(* IEC 61131-3 sources: Dev/Dev_V200/200 (part 8) *)

(* ---- _Nh_MNU.st ---- *)
{ $ IFDEF __NH_WEB }

(*   vyhodnotenie vybrateho menu prebieha

   -  _Nh_Web_CMD (_NhCmd)         - vyvola akciu :
   -  _NhCmdAction   - co sa ma urobit po vybrati volby menu + podporne akcie (ulozi udaje z klasickej web-maker PAGE...)
   -  _NhCmdScreen   - nadefinuje objekty obrazovky + filtre a typ obrazovky (obj)

*)

//********* MNU *******************************************

VAR_GLOBAL
  aWht   : NH_TCH_WHT;
END_VAR

FUNCTION _NhFavNaz {HIDDEN}  : BOOL    // najde aktualne vybraty FAV a zapise veho nazov
   VAR_INPUT
      sav   : BOOL;
   END_VAR
   _NhFavNaz := true;
   FOR nd := 1 TO aCfg[20].rec DO
      _NhxDev(c := 20, n := nd, x:=16);
      xFav := xDev;
      IF xFav^.cx = xA^.fav THEN
         IF sav THEN
            xFav^.cf.Name := xL^.naz;
         ELSE
            xL^.naz := xFav^.cf.Name;
         END_IF;
         nd := 0;
         RETURN;
      END_IF;
   END_FOR;
   _Nh_Lang(id := 18 ,txt := ADR( xL^.naz ), zn:=20);             // oblubene
   nd := 0;
END_FUNCTION

FUNCTION _NhDefSet {HIDDEN}  : BOOL    // vzdy na zaciatku LEN na tomto mieste sa nadefinuju parametre vsetkych browsov, frame....
   VAR_INPUT
      chg      : BOOL;
   END_VAR
   _NhDefSet      := true;
   xU^.o[1]       :=  eMnH.o[1];                                   // aktivuje logo
   IF chg THEN

      xM^.set           := false;

      xUsr^.cx.LastSet  := false;
      CASE xU^.o[2].fn OF
         23:   xU^.o[2].fn := 25;   xM^.set           := true;
                                    xUsr^.cx.LastSet  := true;
         25:   xU^.o[2].fn := 23;
        ELSE   xU^.o[2].fn := 0;
      END_CASE;
   ELSIF xUsr^.cx.Set THEN
      xU^.o[2]       :=  eMnH.o[2];                               // default setup (sivy)
      IF xUsr^.cx.LastSet THEN      //OR aSys.NewDbx THEN
         xM^.set     := true;
         xU^.o[2].fn := 25;
      ELSE
         xM^.set := false;
         xU^.o[2].fn := 23;
      END_IF;
   ELSE
      xU^.o[2].cm := 0;                                              // nezobrazi sa
      xU^.o[2].fn := 0;
      xM^.set     := 0;
   END_IF;
END_FUNCTION

/// *******************************

FUNCTION _Nh_Web_CMD_Screen    : BOOL       // NADEFINUJE OBJEKTY OBRAZOVKY podla akcie od CMD
   (*
    screen sa rozlisuje podla xL^.obj
    - vytvori cistu LVL
    - nadefinuje vrchne a spodne menu
    - v naplni nazov screenu
    - naplni filter DEV (pre brows)
    - naplni filter ROM
    - prelozi nazov do vybrateho jazyka
   *)
   VAR_INPUT
      eMnu     : BOOL;
      obr      : INT;
      obj      : USINT;
      mnu      : USINT := 0;                                               // povolenie menu zmeny DSH (cislo vrchneho menu) 1,2
		n			: USINT;
   END_VAR
   _Nh_Web_CMD_Screen   := 0;
   xM^.wht        := 20;                                                   // pokusi sa najst 1 vetu podla usra
   xL^.brw        := true;
   xL^.obj        := obj;
   xL^.vis        := true;

//   _NhxUsr(u:= xA^.usr);                                                   // namapuje usra
   IF xL^.obj > 30 THEN
      xL^.dsh        := 1;
      mnu            := 0;
   ELSE
      xL^.dsh        := xUsr^.cx.brw[ xL^.obj ];
   END_IF;
   nd             := 0;                                                    // ID textu do xL^.naz

	IF xF^.cf.c > 0 AND xF^.cf.c <> 2 THEN
	   _NhxPt(c := xF^.cf.c, n := xF^.cf.n,x:=47);               				// namapuje hlavicku, napr. koli zisteniu ROM
	END_IF;

   CASE obj OF
     0:  // home page
         mnu            := 0;
         _NhDefSet();
         xL^.vaz        := 1;
         xL^.fvz        := true;
         xU^.o[3].fn   := 0;                                              // zrusi HOME
         xU^.o[8].fn   := 0;                                              // zrusi ON/OFF
         xF^.cf.c      := 3;                                               // default DEV je zon pre cely dom
         xF^.cf.n      := 1;
         xU^.n         := 0;                                               // ziadne vybrate menu
         _NhName(xName := ADR(xL^.Naz) , cf := xF^.cf.c, nd := xF^.cf.n);  //'Môj domov';
         xM^.naz        := xL^.Naz;
         xF^.dev.n[0]   := true;
         xM^.wht        := 25;                                              // pokusi sa najst 1 vetu podla usra
         xL^.dsh        := 0;
         mnu            := 0;

     1: // brow-Zoznam FAV
            nd             := 19;                                          // cislo textu v _NhLang
            xF^.dev.n[20]  := 1;
            xU^.o[2].fn    := 32;                                          // +
            xU^.o[2].cm    := 101;                                          // pridat oblubeny do zoznamu usra
            xF^.cf.c       := 20;                                               // default DEV je zon pre cely dom
            xL^.dsh        := 1;
            mnu            := 0;

     2: // brow-FVL
            _NhFavNaz();
            xF^.dev.n[0]   := 1;
            xL^.vaz        := 1;                                           // cislo vazby
//            xL^.fvz        := true;
            xF^.cf         := xA^.fav;

     3:  // brow-Quick (FAV)
            _NhFavNaz();
            xF^.dev.n[0]   := 1;
            xL^.vaz        := 1;
//            xL^.fvz        := true;
            xF^.cf         := xA^.fav;

     4: // brow-DASH (FAV)
            _NhFavNaz();
            xF^.dev.n[0]   := 1;
            xL^.vaz        := 1;
//            xL^.fvz        := true;
            xF^.cf         := xA^.fav;

     5: // brow-Rooms
            nd             := 7;
            xF^.cf.c       := 1;
            xF^.dev.n[1]   := 1;
            IF xA^.admin THEN
               xU^.o[2].fn    := 32;                                       // pridat ROM
               xU^.o[2].cm    := 101;
            END_IF;
            mnu   := 0;

     6: // brow-ZONES
            nd             := 8;
            xF^.cf.c       := 3;
            xF^.cf.n       := 0;
            xL^.dsh        := 1;
            mnu            := 0;
            IF xA^.admin THEN
               xU^.o[2].fn    := 32;                                       // pridat zonu
               xU^.o[2].cm    := 101;
               _NhFilDev(wht:=2, row:=201);
            ELSE
               _NhFilDev(wht:=2, row:=200);
            END_IF;

     7: // brow-CAT
            IF xU^.o[6].wh = 24 THEN
               xF^.typ        := -2;   									// setup menu
               nd             := 12;
	            IF xM^.set THEN
   	            xU^.o[2].fn    := 230;                         	// save
      	         xU^.o[2].cm    := 101;
	            END_IF;
            ELSE
               xF^.typ        := -1;                              // odfiltruje kategorie na 1.urovni  (xCid^.typ=1);
               nd             := 9;
            END_IF;
            xF^.cf.c          := 2;
//            xF^.dev.n[2]      := 1;

     8: // brow-ACT
            nd             := 10;
            xF^.cf.c       := 5;
            xF^.dev.n[2]  	:= true;											// povoli kategorie
            xF^.dev.n[5]   := 1;
//            xF^.cat.n[54]  := 1;											// + DALI SCENY
            IF xM^.set THEN
               xU^.o[2].fn    := 32;                           // pridat akciu
               xU^.o[2].cm    := 101;
	            xF^.cat.n[55]  := true;									// + Akcie PSN
            END_IF;
            mnu := 0;

     9: // brow-SCN
            nd             := 11;
            xF^.cf.c       := 4;
            xF^.dev.n[4]   := true;                              	// len sceny
            xF^.dev.n[2]  	:= true;											// povoli kategorie
//            xF^.cat.n[53]  := true;											// + NH SCENY
            xF^.cat.n[54]  := true;											// + DALI SCENY

            IF xM^.set THEN
               xU^.o[2].fn    := 31;                           // pridat scenu
               xU^.o[2].cm    := 101;
            END_IF;
            mnu := 0;

    10: // brow- 1 miestnost
				IF xL^.psn THEN
	            xU^   := xM^.mnu[0];                           // ak pride vnorenim z psn nastavi menu z domceka
				END_IF;
            xU^.n             := 5;                            // cislo vybrateno menu
            xU^.o[xU^.n].wh   := 18;                           // 1.miestnost sive
            xU^.o[xU^.n].fn   := 16;                           // miestnosti biele
            xF^.rom           := INT_TO_USINT(xF^.cf.n);       // filtrovanie 1.miestnosti
            IF xDev^.cf.typ = 0 THEN                        	// 0=len pre administratora, setup miestnost, kde su vsetky co nemaju room
               _NhFilDev(wht:=1, row:=203);
//               xF^.dev.n[43] := false;                           // v setup sa zobrazuju DLs a DLg, tie su v DALI
//               xF^.dev.n[44] := false;
            ELSE
//               xF^.rom           := INT_TO_USINT(xF^.cf.n);       // filtrovanie 1.miestnosti
               IF xM^.set THEN
                  _NhFilDev(wht:=1, row:=_Nh_U12(xA^.admin,204,201));
                  IF xDev^.cf.typ < 10 THEN
                     xU^.o[2].fn := 31;
                     xU^.o[2].cm := 101;                              // pridat scenu
                  END_IF;
                  mnu         := 0;                               // zmenit dash vlavo
               ELSE
                  _NhFilDev(wht:=1, row:=200);
                  mnu            :=  0;
               END_IF;
            END_IF;

    11: // brow - 1 zona
            xU^.n             := 5;                                     // cislo vybrateno spodneho menu
            xU^.o[xU^.n].wh   := 22;
            xU^.o[xU^.n].fn   := 20;
            xF^.dev 				:= eFilt_LIST;                             // empty filter
            xF^.dev.n[1]	 	:= true;
//            xF^.dev.n[22] := true;                          // users
            IF xF^.cf.n = 1 THEN
               xF^.rom := 0;
            ELSE
               xF^.rom := INT_TO_USINT(xF^.cf.n);
            END_IF;

    12: // brow - 1.kategoria
            IF xU^.n = 0 THEN                                           // cislo vybrateno menu

				ELSE
					xU^.n    			:= 6;                                      	// vyberie menu CAT
               xU^.o[xU^.n].fn  	:= 13;                               // nastavi obr 1.CAT sivy
               xU^.o[xU^.n].wh  	:= 13;                               // nastavi obr 1.CAT sivy
				END_IF;
            xF^.rom        := 0;
            xF^.typ        := INT_TO_SINT(xF^.cf.n);
				_NhFilDev(wht:=0);													// vymaze filter DEV,CAT
            xF^.dev.n[2]   := true;												// vsetky CAT
            _NhxRoW(nbr:=xA^.sbj, zon:=true);                        // namapuje xRow na Domcek alebo ak sa pouzivaju subjekty tak na subjekt-byt
				_Nh_Set_ONOFF(set:=xRoW^.cat[ xF^.cf.n ]);

(*
				xU^.o[1].fn   	:= 1;													// NH
 				xU^.o[1].wh   	:= 1;
				xU^.o[1].cm   	:= 24;                            			// menu NH
*)
            mnu         := 0;
            IF xM^.set THEN
               CASE xF^.cf.n OF
                  3:    // Tienenie = ROL
			 					xU^.o[1].fn   	:= 0;
		 						xU^.o[1].wh   	:= 0;
								IF xM^.set THEN
									xU^.o[2].fn   	:= 45;										// sivy COPY
				 					xU^.o[2].cm   	:= 129;                            	// zmena siveho copy na zlty
								ELSE
									xU^.o[2].fn   	:= 0;
				 					xU^.o[2].cm   	:= 0;
								END_IF;
								mnu 				:= 1;

_Nh_Set_ONOFF(set:=false);

				      4:    // vetranie
                        _Nh_Set_ONOFF(set:=false);
                        IF xM^.set THEN
                           xU^.o[2].fn := 339;                                // pridat regulator
                           xU^.o[2].cm := 101;                                // pridat regulator akcia
                        ELSE
                           xU^.o[2].fn := 0;                                // pridat regulator
                        END_IF;

                  5:    // KOMFORT : dodefinuje pridanie regulatora
                        _Nh_Set_ONOFF(set:=false);
                         xU^.o[2].fn := 182;                                // pridat regulator
                         xU^.o[2].cm := 101;                                // pridat regulator akcia

                  7:    // brany
                        _Nh_Set_ONOFF(set:=false);										// bran nie je vela, NEnastavi sa filter
//                        mnu            := 1;
                  39:    // setup HET
								_Nh_Set_ONOFF(set:=false);
                        IF xA^.admin THEN
	                         xU^.o[2].fn := 225;                                // pridat vsetky regulatory
   	                      xU^.o[2].cm := 141;                                // pridat regulator akcia
								END_IF;
(*

                 44:    // vsetky dev bez miestnosti alebo zle priradene
                        _NhFilDev(wht:=1, row:=199);

//                        xF^.dev     := _NhfDev.rom[199];                // zoznam DEV pri rezime SET
                        xU^.o[6].wh    := 11;                                                 // default prave horne menu je nic
                        xU^.o[6].cm    := 34;
                        xU^.o[6].fn    := 10;                                                 // default prave horne menu je nic                                                                         // default prave horne menu je nic
                        xL^.obj        := 13;
//                        xL^.fdv        := 0;
//                        mnu            := 1;
*)
                  41:   //

               ELSE
               END_CASE;
            END_IF;
		   	rb:=_Nh_FRM_Read(frm:=232);     						// CAT
  	         nd := yFrm_232.cat[xF^.cf.n].txt;                                  	// hlavny text {druhy riadok je vzdy o cislo vacie"
            xL^.dsh     := 1;

(*
            xU^.n    := 6;                                           // cislo vybrateno menu
            IF xU^.o[xU^.n].wh  <>  24 THEN                          // setup zostava
               xU^.o[xU^.n].fn  := 13;
               xU^.o[xU^.n].wh  := 13;
               xU^.o[3]       := eMnH.o[3];                                     // aktivuje HOME
            END_IF;
            xU^.o[2].fn    := 0;                                                 // default prave horne menu je nic
            xU^.o[2].cm    := 0;
            xF^.rom        := 0;
            xF^.typ        := INT_TO_SINT(xF^.cf.n);
*)

    13:  // brow - vsetky zony pre SEC

(*

            xL^.psn  := true;
            xU^.n    := 6;                                           // cislo vybrateno menu
            IF xU^.o[xU^.n].wh  <>  24 THEN                          // setup zostava
               xU^.o[xU^.n].fn  := 13;
               xU^.o[xU^.n].wh  := 13;
               xU^.o[3]       := eMnH.o[3];                                     // aktivuje HOME
            END_IF;
            xU^.o[2].fn    := 0;                                                 // default prave horne menu je nic
            xU^.o[2].cm    := 0;
//            xF^.dev.n[2]   := true;
            xF^.rom        := 0;
            xF^.typ        := INT_TO_SINT(xF^.cf.n);
//            nd             := _NhDefCat[xF^.cf.n].ID;
//            xL^.dsh        := xUsr^.cx.brw[ xL^.obj ];
            mnu            := 2;
*)

    14:  // brow - 1 zona SEC
            xL^.psn           := true;
            xU^.n             := 5;                                     // cislo vybrateno menu
            xU^.o[xU^.n].wh   := 22;
            xU^.o[xU^.n].fn   := 20;
            xU^.o[2].fn       := 0;
            xF^.dev.n[1]      := true;                            // zobrazuju sa len mistnosti, ktore vstupuju do zony
            xF^.rom           := 0;
//            xL^.dsh           := xUsr^.cx.brw[ xL^.obj ];
            mnu               := 0;

    15: // brow- 1.miestnost zobrazuje len SEC
//            xL^.psn           := true;
            xU^.n             := 5;                            // cislo vybrateno menu
            xU^.o[xU^.n].wh   := 18;                           // 1.miestnost sive
            xU^.o[xU^.n].fn   := 16;                           // miestnosti biele
            xF^.rom           := INT_TO_USINT(xF^.cf.n);       // filtrovanie miestnosti
//            xL^.fRom          := true;
            _NhFilDev(wht:=1, row:=202);
//            xF^.dev           := _NhfDev.rom[202];                // zoznam DEV pri rezime SET
//            xL^.dsh           := xUsr^.cx.brw[ xL^.obj ];
            mnu               := 2;

    20: // brow-BLK
            nd             := 107;
            xF^.cf.c       := 35;
            xF^.dev.n[35]  := 1;
            IF xM^.set THEN
               xU^.o[2].fn    := 195;                           // + BLK
               xU^.o[2].cm    := 101;
            END_IF;

    21: // brow-TIM
            nd             := 333;
            xF^.cf.c       := 50;
            xF^.dev.n[50]  := 1;
            IF xM^.set THEN
               xU^.o[2].fn    := 294;                           // + TIM
               xU^.o[2].cm    := 101;
            END_IF;

    22: // brow-SMW
            nd             := 339;
            xF^.cf.c       := 25;
            xF^.dev.n[25]  := 1;
            IF false THEN // xM^.set THEN
               xU^.o[2].fn    := 299;                           // + SMW
               xU^.o[2].cm    := 101;
            END_IF;

    30: // brow priradenie ROM/KLA do ZON
				xF^.dev 				:= eFilt_LIST;                             // empty filter
(*
				IF n = 7 THEN
	            xF^.dev.n[24] 	:= true;									// len KLAvesnice
            	xU^.n       	:= 7;
            	nd             := 413;									// miestnosti v zone
				ELSE
	            xF^.dev.n[1] 	:= true;									// len ROM
            	xU^.n       	:= 8;
            	nd             := 407;									// miestnosti v zone
				END_IF;
*)
				xPt^.al.lst		:= false;
           	xU^.n       	:= 8;
            xF^.dev.n[1] 	:= true;									// len ROM
	         xU^.o[4].fn    := 0;                           	// vypne CAT
            xL^.fvz    	 	:= true;                      	// default filtruje
	         xU^.o[2].fn    := 0;                           	// vypne +
         	xU^.o[3].fn    := 38;
            mnu            := 0;
            xL^.brw     	:= 1;
            xL^.dsh     	:= 1;                                              // pevny DASH, 1 riadok
            xL^.chk     	:= true;                                           // priznak ze sa zaskrtava CHK, nie FAV
            xL^.vaz     	:= 0;

(*
    31: // akcie LOCK/UNLOCK
				xF^.dev 				:= eFilt_LIST;                             // empty filter
            xF^.dev.n[3] := true;
            xU^.o[4].fn    := 10;
            nd             := 0;

            nd             := 408;									// akcie od alarmu

            mnu            := 0;
            xL^.brw     := 1;
            xL^.dsh     := 1;                                              // pevny DASH, 1 riadok
            xL^.chk     := true;                                           // priznak ze sa zaskrtava CHK, nie FAV
            xL^.vaz     := 2;
            xU^.n       := 5;
*)

    32: // akcie od ALARMU
    			xF^.dev 				:= eFilt_LIST;                             // empty filter
            xF^.dev.n[48] 	:= true;
//            xF^.dev.n[35] 	:= true;
//            xF^.rom 			:= INT_TO_USINT(xF^.cf.n);
            nd             := 408;									// akcie od alarmu
            mnu            := 0;
            xL^.brw     	:= 1;
            xL^.dsh     	:= 1;                                              // pevny DASH, 1 riadok
            xL^.chk     	:= false;                                           // priznak ze sa zaskrtava CHK, nie FAV
            xL^.vaz     	:= 0;
            xU^.n       	:= 6;
            IF xA^.UsrRight > 1 THEN
               xU^.o[2].fn    := 32;                           // pridat akciu
               xU^.o[2].cm    := 101;
            END_IF;

    33: // simulacie pritomnosti
    			xF^.dev 				:= eFilt_LIST;                             // empty filter
            xF^.dev.n[10] 	:= true;
            xF^.dev.n[35] 	:= true;
            nd             := 410;
            mnu            := 0;
            xL^.brw     	:= 1;
            xL^.dsh     	:= 1;                                              // pevny DASH, 1 riadok
            xL^.chk     	:= true;                                           // priznak ze sa zaskrtava CHK, nie FAV
            xL^.vaz     	:= 0;
            xU^.n       	:= 5;
            IF xA^.UsrRight > 1 THEN
               xU^.o[2].fn    := 32;                           // pridat akciu
               xU^.o[2].cm    := 101;
            END_IF;

    47: // brow- dali Sceny
         mnu            := 2;
         _Nh_FRM_Read(frm:=6);
         xF^.dev.n[44]  := 1;
         xU^.o[7].fn := 334;                            // browser DLg  47
         xU^.o[4].fn    := 0;                           // CAT nebude viditelne
         xL^.dsh        := 1;
         xU^.o[3].fn := 35;                                      // bez vazieb aj s
         xU^.o[5].fn := 16;                                      // vsetky ROM
         xU^.o[6].fn := 335;                                     // len jeden master co je v hlavicke
         xU^.o[8].fn := 49;                                      // aj  ON aj OFF

    48: // brow- zoznam SLAVE k MASTRU v hlavicke
         mnu            := 2;
         _Nh_FRM_Read(frm:=6);
         xF^.dev.n[43]  := 1;
         xU^.o[6].fn    := 335;
         xL^.dsh        := 1;
			_Nh_Set_ONOFF(set:=xDev^.al.sta=1);

    49: // brow-DALI - zoznam Master
            nd             := 334;
            xF^.dev.n[42]   := 1;
            xM^.set := true;
            xL^.dsh := 1;

    50: // vstup do VAZIEB cez setup v riadku
            IF eMnu THEN
	            _Nh_FRM_Read(frm:=17);
               IF obr = 0 THEN
                  obr := xU^.o[2].fn;
               END_IF;
//               xU^         := eMvz;                                        // default menu 1
               xU^.o[2].fn := obr;  //_NhObrNbr(cf := xF^.cf.c, t := xDev^.cf.typ);      // default obrazok vyssej casti
					IF aCfg[ xF^.cf.c ].lst = false THEN
//						xU^.o[7].cm	:= 0;
//						xU^.o[7].fn := 0;
					END_IF;
//					xL^.vis		:= false;
            END_IF;
//					IF aCfg[ xF^.cf.c ].Visible = false THEN
//						xU^.o[6].fn	:= 0;
//						xU^.o[6].cm	:= 0;
//   				END_IF

            xU^.n       := 8;                                           // prednastavi LIST-menu
            xL^.obj     := 50;
            xL^.brw     := 1;
            xL^.dsh     := 1;
            xL^.chk     := true;                      // priznak ze sa zaskrtava CHK, nie FAV
				xL^.vaz     := 2;
				xL^.fvz     := xPt^.al.vaz;					// ak ma vazby, nastavi sa filter
            mnu 			:= 0;                         // nevybera sa DSH
            IF xL^.fvz THEN									// ak je zapnuty filter, vypne filtrovanie ROM
            	xF^.rom  := 0;
     	      ELSE
     	      	xF^.rom  := xPt^.cf.rom;
           	END_IF;
//            _Nh_Vaz_ROM();
//            _Nh_Vaz_DEV();
				_Nh_Vaz_DEV();
            _Nh_Vaz_CHK();

    51: // vstup do DEV-listu.	moze vzniknut xL^.obj :=     43 Dls, 44 DLg v hlavicke
            IF eMnu THEN
	            _Nh_FRM_Read(frm:=17);
               IF obr = 0 THEN
						_NhTypObr(cf:=xF^.cf.c, typ:=xPt^.cf.typ);
						obr := xObrWht^.obr;
               END_IF;
               xU^.o[2].fn := obr;
               xL^.chk     := true;                                     // priznak ze sa zaskrtava CHK, nie FAV
               xL^.brw     := 1;
               xL^.dsh     := 1;                                        // pevny DASH, 1 riadok
					xL^.vis		:= false;
            END_IF;
				xL^.vaz     := 0;
				IF xU^.o[6].cm	= 77 OR xU^.o[6].cm	= 75 THEN 		// Ext.vazby OR RGBWA
					xL^.vis		:= false;
					xU^.o[6].fn	:= xU^.o[6].fn;
				ELSIF xU^.o[6].cm	= 36 THEN //aCfg[ xF^.cf.c ].Visible  THEN
					xU^.o[6].fn	:= _Nh_O12(in := xL^.vis , o1:=113, o2:=112);
				ELSIF aCfg[ xF^.cf.c ].Visible THEN
					xU^.o[6].fn	:= 112;
					xU^.o[6].wh	:= 113;
					xU^.o[6].cm	:= 36;
					xU^.o[6].fn	:= _Nh_O12(in := xL^.vis , o1:=113, o2:=112);
				ELSE
					xU^.o[6].fn	:= 0;
					xU^.o[6].cm	:= 0;
				END_IF;
            xL^.fvz     := xPt^.al.lst;
            xU^.n       := 7;                                           // prednastavi LIST-menu
            IF xL^.fvz THEN
               xF^.rom  		:= 0;
               xF^.dev.n[1]	:= 1;    											// vsetky dev
               xL^.fdv			:= 0;  	                               	// vsetky CAT
            ELSE
               xF^.rom  := xPt^.cf.rom;
            END_IF;
            mnu 			:= 0;
				ok				:= false;
            CASE xF^.cf.c OF
              4 : // SCN-LIST
                  xL^.vaz     	:= 3;
              5 : // ACT-LIST
                  xL^.vaz     	:= 4;
              6 : // HET-reg
                  xL^.vaz     	:= 4;
						;
              7 : // KOT-teplota
						;
              8 : // TVE-teplota
						;
              9 : // CER
						;
             47 : // HEV-reg
                  xL^.vaz     	:= 4;
             35 : // BLK-LIST
                  xL^.vaz     	:= 4;
             37 : // GATE-koncovy snimac DOOR/WIN
                  xL^.vaz     := 0;
             43 : // DLS-Dali-DEV LIST - len dali sceny do ktorych DLs patri
             		xL^.obj  		:= 43;
                  xL^.vaz  		:= 0;
						xDLs				:= xPt;
						xF^.dev.n[44] := true;
						{$IFDEF __NH_DALI}
		            xL^.fvz     := xDLs^.cx.scn.grp <> _eBtn15;
                  {$END_IF}
		            IF xL^.fvz THEN
      		         xF^.rom  := 0;
		            ELSE
      		         xF^.rom  := xPt^.cf.rom;
            		END_IF;
						xPt^.al.lst 	:= false;			// resetne zobrazovanie pouzitej sceny (siva farba pod cislom sceny)
						IF xDls^.cx.cfg.out5inOne THEN								// do TVE, bude zobrazena RGBWA +
							xU^.o[6].fn	:= 124;
							xU^.o[6].wh	:= 125;
							xU^.o[6].cm	:= 75;
						END_IF;

             44 : // DLg-LIST : v hlavicke je DALI scena (DLg), v liste su len DLs  DLg->DLs
						{$IFDEF __NH_DALI}
                  xL^.obj     			:= 44;
						xDLg						:= xPt;
						xDLg^.cx.sta.Present := false;			// resetne zobrazovanie pouzitej sceny (siva farba pod cislom sceny)
                  xU^.o[4].fn := 0;          				// CAT sa pri DLg nezobrazuju, mozu byt len DLs
						xPt^.al.lst 			:= false;			// resetne zobrazovanie pouzitej sceny (siva farba pod cislom sceny)

                  {$END_IF}
             48 : // ALA
                  xL^.vaz     := 4;
            ELSE  // v hlavicke je klasicke DEV avaz[3], alebo DEV-ballast - ma svoju strukturu scn

//                  xL^.vaz     := 3;          // dali sceny maju vazby len k DLs
            END_CASE;
				_Nh_Vaz_DEV();
            _Nh_Vaz_CHK(ini:=true);

	 52: 	// vstup do menu - SETUP - priradeneie do ROM/ZON

            xL^.fvz     	:= 0;
            xL^.chk     	:= 1;                                           // priznak ze sa zaskrtava CHK, nie FAV
            xL^.dsh     	:= 1;
  	 			xL^.vaz     	:= 0;
            xF^.dev.n[1]  	:= true;
				IF xL^.obj <> 70 THEN
	            _Nh_FRM_Read(frm:=54); 										// nacita menu
					IF aCfg[xF^.cf.c].zone THEN
		            xF^.dev.n[3]  	:= 1;
					END_IF;
//	           	xU^.o[2].fn 	:= _NhObrNbr(cf := xF^.cf.c, t := xDev^.cf.typ);      // default obrazok vyssej casti
					_NhTypObr(cf:=xF^.cf.c, typ:=xPt^.cf.typ);
					xU^.o[2].fn := xObrWht^.obr;

//					IF xDev^.cf.rom > 0 THEN
					IF xPt^.cf.rom > 0 THEN
		            xL^.fvz     	:= 1;
					END_IF;
				END_IF;
//            xU^.n       	:= 8;
				xL^.obj     	:= 70;							// aj rom , u niektor aj ZON
            mnu 				:= 0;
				_Nh_Vaz_CHK();

    55: // Extrne vazby DEV - na DALI,MQTT,....
				xL^.vaz     := 0;
            IF eMnu THEN
	            _Nh_FRM_Read(frm:=17);
               IF obr = 0 THEN
//                  obr := _NhObrNbr(cf := xF^.cf.c, t := xPt^.cf.typ);      // default obrazok vyssej casti;
						_NhTypObr(cf:=xF^.cf.c, typ:=xPt^.cf.typ);
						obr := xObrWht^.obr;

               END_IF;
               xU^.o[2].fn := obr;
               xL^.chk     := true;                                     // priznak ze sa zaskrtava CHK, nie FAV
               xL^.brw     := 1;
               xL^.dsh     := 1;                                        // pevny DASH, 1 riadok

					xU^.o[6].fn	:= 367;
					xU^.o[6].wh	:= 368;
					xU^.o[6].cm	:= 77;
					n				:= 6;

(*
					xU^.o[7].fn	:= 367;
					xU^.o[7].wh	:= 368;
					xU^.o[7].cm	:= 77;
					n				:= 7;
*)

            END_IF;
            xU^.n       := n;                                           // prednastavi LIST-menu
//				xL^.vis		:= false;
            mnu 			:= 0;
				ok				:= false;
            CASE xF^.cf.c OF
              6 : // HET
						xHet		:= xPt;
              7 : // KOT
						xTve		:= xPt;

              8 : // TVE
						xTve		:= xPt;

              9 : // CER
						xTve		:= xPt;
(*
             43 : // DLS-Dali-DEV LIST - len dali sceny do ktorych DLs patri
						xDLs := xPt;
						IF xDls^.cx.cfg.out5inOne THEN								// do TVE, bude zobrazena RGBWA +
							xU^.o[6].fn	:= 124;
							xU^.o[6].wh	:= 125;
							xU^.o[6].cm	:= 75;
						END_IF;
						xF^.dev.n[43] := true;
*)
            ELSE  // v hlavicke je klasicke DEV avaz[3], alebo DEV-ballast - ma svoju strukturu scn
					;
            END_CASE;
				_Nh_Vaz_DEV();
            _Nh_Vaz_CHK(ini:=true);

    56: // list RGBWA je DLs v hlavicke
            IF eMnu THEN
	            _Nh_FRM_Read(frm:=17);
               xU^.o[2].fn := obr;
               xL^.chk     := true;                                     // priznak ze sa zaskrtava CHK, nie FAV
               xL^.brw     := 1;
               xL^.dsh     := 1;                                        // pevny DASH, 1 riadok
					xL^.vis		:= false;
					xL^.fvz 		:= true;

					xU^.o[6].fn	:= 124;
					xU^.o[6].wh	:= 125;
            END_IF;
            xU^.n       		:= 6;                                           // prednastavi LIST-menu
				xL^.vaz     		:= 0;
				_Nh_Vaz_DEV();
            _Nh_Vaz_CHK();

(*
    56: // brow-MSG (all)
            nd             := 56;
            xF^.cf.c       := 46;
            xF^.dev.n[46]  := 1;
            mnu            := 1;
            IF xM^.set THEN
               xU^.o[2].fn    := 237;                           // pridat akciu
               xU^.o[2].cm    := 101;
	            xF^.cat.n[57]  := true;									// + Akcie PSN
            END_IF;
*)

    57: // brow-MSG (len alarm)
            nd             := 388;
            xF^.cf.c       := 46;
            xF^.dev.n[46]  := 1;
            mnu            := 1;

    60: // brow - uzky vyber pre kopirovanie POI: ROM/HET/VEN
           	_Nh_FRM_Read(frm:=79);							// menu kopirovania
            xF^.dev.n[xF^.cf.c]  := true;                    	// filter na CF podla hlavicky
				xL^.naz 					:= xPt^.cf.Name;					// nazov dev z ktoreho sa kopiruje
            xL^.dsh 					:= 4;                         // tenky browser

(*
   100: // Dashboard meteostanica

         xL^.obj        := 205;                                      // podhodi sa 200
         xA^.tch.cm     := 206;
         xA^.tch.cmd    := 206;                                      // vrati sa uz do 200
			_Nh_FRM_Read(wht := 3, frm :=  69);
         xF^.rom        := 0;                                      // podla tohto sa nadefinuje menu
			xF^.cf.c			:= 3;
			xF^.cf.n			:= 1;
			nd					:= 240;
			mnu				:= 0;

      _NhLang(id := nd ,txt := ADR( xL^.naz ));

   xM^.wht        := 0;                                                   // pokusi sa najst 1 vetu podla usra
   xL^.brw        := 0;
//   xL^.obj        := obj;
   xL^.vis        := 0;
*)

   END_CASE;
   IF mnu > 0 THEN
      _Nh_Brw_Dsh_Chg(mnu := mnu);
   END_IF;
   IF nd > 0 THEN
      _Nh_Lang(id := nd ,txt := ADR( xL^.naz ),zn:=20);
   END_IF;

END_FUNCTION

FUNCTION _NhxLvl {HIDDEN}  : BOOL
   i     := xM^.lvl;
   xL    := ADR(xM^.lvd[i]);                                // old Level
   xF    := ADR(xL^.fil);
   xU    := ADR(xM^.mnu[i]);
END_FUNCTION

FUNCTION _NheLvl  {HIDDEN}   : BOOL                                // dopredu,dozadu
   VAR_INPUT
      lvl      : SINT;
   END_VAR
   _NheLvl 		:= true;
   CASE lvl OF
     1 : // o uroven dopredu
         IF xM^.lvl < 3 THEN
            xM^.lvl     := xM^.lvl + 1;                        // zvysi sa lvl
            _NheBrw(wht := 3);                                 // vymaze sa veta lvd[lvl] (nie data ani riadok odkial odskok je)
            _NhxLvl();                                         // namapuju sa k novemu lvl

//            xB^.r[0]    := xR^;                             // v r[0] bude cela veta a odial r[0].h.chk - ci bola vazba

            xU^         := xM^.mnu[xM^.lvl-1];                 // na zaciatok sa preberie menu
            xU^.o[1].fn := 6;                                  // sipka spat
            xU^.o[1].cm := 31;                                 // cmd spat
            xL^.vis     := xM^.lvd[xM^.lvl-1].vis;
            xL^.psn     := xM^.lvd[xM^.lvl-1].psn;

            // preberu sa udaje z riadka do pomocnej struktury
            IF xR^.h.chk THEN
               yIO      := xR^.o.ob[4].cf;                     // pre detail aby sme vedeli vazby
            ELSE
               yIO      := xR^.h.cf;
            END_IF;
            IF xR^.h.chk AND xA^.tch.obj = 4 THEN              // v zaskrtnutej vazbe sa ide do properties vyssej casti
               yIO      := xR^.h.cf;
               xF^.cf   := xR^.o.ob[4].cf;                     // hlavicka sa preberie z vyssej casti s parametrom v riadku
               IF xA^.tch.cmd = 200 OR xA^.tch.cmd = 204 THEN

//                  xL^.vaz   := xR^.h.cf.c;                     //**-** ak sa ide z vazby, zapamata sa cf z vazby

               END_IF;
            ELSE
               xF^.cf   := xR^.h.cf;                           // hlavicka sa preberie z riadka
            END_IF;
            IF xF^.cf.c <> 2 THEN                              // nazov u CAT sa zoberie priamo z textov
               _NhName(xName := ADR(xL^.naz) , cf := xF^.cf.c, nd := xF^.cf.n);
            END_IF;

            xA^.tch.Q    := false;                              // pri vstupe do noveho LVL sa resetuje sa priznak stlacenia nad objektom
            xA^.tch.Qr   := false;                              // pri vstupe do noveho LVL sa resetuje sa priznak stlacenia nad objektom
            xA^.tch.Qf   := false;                              // pri vstupe do noveho LVL sa resetuje sa priznak stlacenia nad objektom
         ELSE
            xM^.wht     := 10;
            _NheLvl     := false;
         END_IF;

    -1: // o uroven spat
			aSys.RefCycNew := 1;															// pri vsupe/spat sa urobi refresh
   		_NheBrw(wht := 9);                                 	// vymaze pod = editacia TypeDay
         IF xM^.lvl > 0 THEN
            xM^.lvl   := xM^.lvl - 1 ;
         ELSE
            xM^.lvl   := 0 ;
         END_IF;
         _NhxLvl();
         xM^.wht     := 25;                                    // od 1.zapamataneho riadku
    -2: // o uroven spat
			aSys.RefCycNew := 1;															// pri vsupe/spat sa urobi refresh
   		_NheBrw(wht := 9);                                 	// vymaze pod = editacia TypeDay
         IF xM^.lvl > 1 THEN
            xM^.lvl   := xM^.lvl - 2 ;
         ELSE
            xM^.lvl   := 0 ;
         END_IF;
         _NhxLvl();
         xM^.wht     := 25;                                    // od 1.zapamataneho riadku

     3 : // o uroven dopredu
         xM^.lvl     := xM^.lvl + 1;                        // zvysi sa lvl
         _NheBrw(wht := 3);                                 // vymaze sa veta lvd[lvl] (nie data ani riadok odkial odskok je)
         _NhxLvl();                                         // namapuju sa k novemu lvl
     4 : // o uroven dopredu , ponecha data pre kopirovanie
         IF xM^.lvl < 3 THEN
	         yIO      := xF^.cf;
   	      xM^.lvl     := xM^.lvl + 1;                        // zvysi sa lvl
      	   _NheBrw(wht := 8);                                 // vymaze sa veta lvd[lvl] (nie data ani riadok odkial odskok je)
         	_NhxLvl();                                         // namapuju sa k novemu lvl
	         xF^.cf   := yIO;                           			// hlavicka sa preberie z riadka
			END_IF;
   ELSE                                                        // v tej istej urovni
         _NheBrw(wht := 3);                                 // vymaze sa veta lvd[lvl] (nie data ani riadok odkial odskok je)
         _NhxLvl();                                         // namapuju sa k novemu lvl
         // preberu sa udaje z riadka do pomocnej struktury
         yIO      := xR^.h.cf;
         xF^.cf   := xR^.h.cf;                           // hlavicka sa preberie z riadka
         _NhName(xName := ADR(xL^.naz) , cf := xF^.cf.c, nd := xF^.cf.n);
   END_CASE;
END_FUNCTION

FUNCTION _NhWebSave  {HIDDEN} : BOOL    // prestavi menu vazieb aj suvisiacich filtrov
   VAR_INPUT
      NoLvl    : BOOL;
   END_VAR
   _NhWebSave  := true;
   IF xF^.cf.c > 0 THEN
      _NhxDev2(c := xF^.cf.c, n := xF^.cf.n, x:=17);
      CASE xF^.cf.c OF
         22 :  xUsr2  := xDev2;
               IF xF^.cf.n = 1 THEN
                  yUSR.cf.blk    := 0;                                  // admin si nemoze prepisat sbj z 0
						xA^.admin 		:= 1;
					ELSE
						xA^.admin 		:= 0;
               END_IF;
               xUsr2^  			:= yUsr;
					xA^.UsrRight 	:= xUsr2^.cx.UsrRight;

(*
               IF xF^.cf.n = 1 THEN
//                  yUSR.cf.sbj       := 0;                                  // admin si nemoze prepisat sbj z 0
                  yUSR.cf.blk       := 0;                                  // admin si nemoze prepisat sbj z 0
//                  yUSR.cx.UsrRight  := 2;                                  // admin si nemoze prepisat sbj z 0
               END_IF;
               IF xUsr^.cx.UsrRight = 2 THEN
                  xUsr2^  := yUSR;
               ELSIF xUsr^.cx.UsrRight = 1 THEN                      // superuzivatel
                  IF yUSR.cx.UsrRight > 1 THEN
                     yUSR.cx.UsrRight := 1;
                  END_IF;
//                  yUSR.cf.sbj := xUsr^.cf.sbj;                       // nemoze subjekt
                  xUsr2^      := yUSR;
               ELSIF xF^.cf.c = xA^.usr THEN                         // uset moze opravit len sam seba
                     xUsr2^.cf.Name       := yUSR.cf.Name;
                     xUsr2^.cx.mail       := yUSR.cx.Mail;
                     xUsr2^.cx.gsm        := yUSR.cx.gsm;
                     xUsr2^.cx.KeyPas     := yUSR.cx.KeyPas;
                     xUsr2^.cx.LoginHome  := yUSR.cx.LoginHome;
               END_IF;
*)
      END_CASE;
   END_IF;
   IF NoLVL = false THEN
      _NheLvl( lvl := -1 );                                              // o LVL dopredu
   END_IF;
   xM^.frm := false;
   xM^.htx := 0;
   xM^.htt :=  '';
END_FUNCTION

FUNCTION  _Nh_Web_CMD_Action       : BOOL  // _NhObrMnu NADEFINUJE HOME SCREEN, VYVOLA AKCIU PO STLACENI MENU/DASH, TIEZ ulozi udaje z klasickej web-maker PAGE
   (*
   - uplne na zaciatku nadefunuje HOME screen (pre kazdy subjekt iny)
   - ak je aktivna klasicka webmaker-page s editaciou premennych, ulozi tieto premenne
   - zisti sa stlacenie menu vrchneho, spodneho, niektoreho s dashboardu v HOME-screen
   - ina akcia je pri stlaceni toho isteho menu, ktore je prave aktivne, a ina pri novej volbe
   - pri stlaceni dashboardu, v HOME sa vyvola prislusna kategoria
   - podla vysledneho vyhodnotenia sa vacsinou prepne / nadefinuje nova obrazovka
   *)
   VAR_INPUT
      mnu      : USINT;
   END_VAR
   _Nh_Web_CMD_Action      := true;
   IF xM^.htx > 0 THEN                                           // ak je nejaky frame
      _NhWebSave(NoLvl := true);                                 // ulozi ak je co
   END_IF;
   rb          := xM^.lvl = 0;                                          // ovplyvni prepinaju volby nad tym istym tlacitko, ked sa vracia z inej urovni, neprepina sa
   xM^.lvl     := 0 ;
   _NhxLvl();
   IF xM^.naz = '' THEN                                                 // uplne nove prihlasenie
      _NheBrw( wht:=1 );
      mnu         := 0;
      xU^         := eMnH;                                              // prida prvotne ciste mnu
      _NhUsrPar( fav := 1);
      xM^.set     := xUsr^.cx.set OR xA^.usr = 1 OR aSys.NewDbx;
      xM^.srt     := xM^.set;
   ELSE
      _NheBrw( wht := 6);                                         // vsetky lvl aj brw
   END_IF;
   xL^.vis     := true;
   IF mnu = 0 THEN                                                      // HOME page
      _Nh_Web_CMD_Screen(obj := 0);
      RETURN;
   ELSIF mnu = xU^.n AND rb THEN                           // vybrate to iste menu v zakladnom leveli = prepnut
      CASE mnu OF
        4  :  // FAV
               CASE xU^.o[mnu].fn OF
                 41: xU^.o[mnu].fn := 59;                   // z FAV na FAV list
                     xU^.o[mnu].wh := 60;
                 59:                                        // prepnutie zo zoznamu FAV
                        CASE xA^.fav.n  OF
                          -1 :   xU^.o[mnu].fn := 199;        // DASH
                                 xU^.o[mnu].wh := 199;
                          -2 :   xU^.o[mnu].fn := 198;        // QUICK
                                 xU^.o[mnu].wh := 198;
                        ELSE     xU^.o[mnu].fn := 41;          // vybraty FAV
                                 xU^.o[mnu].wh := 42;
                        END_CASE;
                  ELSE
                     xU^.o[mnu].fn := 59;
                     xU^.o[mnu].wh := 60;
               END_CASE;
        5  :  // ROOMS
               CASE xU^.o[mnu].fn OF
                 16: xU^.o[mnu].fn := 20;                   // z romms na zone
                     xU^.o[mnu].wh := 21;
                 20: xU^.o[mnu].fn := 16;                   // zo zone na rooms
                     xU^.o[mnu].wh := 17;
               END_CASE;
        7  :  // ACT
               IF xM^.set = false THEN
                  CASE xU^.o[mnu].fn OF
                    27: xU^.o[mnu].fn := 29;                   // z ACT na SCN
                        xU^.o[mnu].wh := 30;
                    29: xU^.o[mnu].fn := 27;                   // SMW->ACT
                        xU^.o[mnu].wh := 28;
                  END_CASE;
               ELSE
                  CASE xU^.o[mnu].fn OF
                    27: xU^.o[mnu].fn := 29;                   // z ACT na SCN
                        xU^.o[mnu].wh := 30;
                    29: xU^.o[mnu].fn :=196;                   // SCN->BLK
                        xU^.o[mnu].wh :=197;
                   196: xU^.o[mnu].fn :=295;                   // BLK->TIM
                        xU^.o[mnu].wh :=296;
(*
                   295: xU^.o[mnu].fn :=235;                   // TIM->MSG
                        xU^.o[mnu].wh :=236;
                   235: xU^.o[mnu].fn := 27;                   // MSG->ACT
                        xU^.o[mnu].wh := 28;
*)
(*
                   295: xU^.o[mnu].fn :=297;                   // TIM->SMW
                        xU^.o[mnu].wh :=298;
                   297: xU^.o[mnu].fn := 27;                   // SMW->ACT
                        xU^.o[mnu].wh := 28;
*)
						 ELSE
                   		xU^.o[mnu].fn := 27;                   // BLK->TIM
                        xU^.o[mnu].wh := 28;
                  END_CASE;
               END_IF;
      END_CASE;
   ELSIF xU^.n = 0 THEN                                     // je aktivne HOME page
      IF mnu = 1 THEN
         xU^.o[6].wh := 24;   										// do spodneho menu cat nastavi setup
         mnu         := 6;                                  // vyberie cas = setup
      ELSE
         xU^.o[6].wh := 11;
      END_IF;
   ELSE
      CASE xU^.o[xU^.n].wh OF
        18  :  // jedna miestnost - vrati na miestnosti
               xU^.o[xU^.n].fn := 16;           // miestnosti siva
               xU^.o[xU^.n].wh := 17;           // miestnosti biela

        22  :  // jedna zona      - vrati na zony
               xU^.o[xU^.n].fn := 20;           // zona siva
               xU^.o[xU^.n].wh := 21;           // zona biela
        24  :  // setup z ikony NH
               xU^.o[xU^.n].fn := 10;           // siva CAT
               xU^.o[xU^.n].wh := 11;           // zona biela
      ELSE
      ;
      END_CASE;
   END_IF;
   xU^.n          := mnu;                       // cislo menu, ktore bude vybrate
   xU^.o[1].fn    :=  0;                                            // zrusi LOGO
   xU^.o[2].fn    :=  0;                                            // zrusi SETUP
   xU^.o[3]       := eMnH.o[3];                                     // aktivuje HOME
   IF xU^.o[8].fn = 0 THEN                                          // prislo sa z HOME
      xU^.o[8]    := eMnH.o[8];                                     // aktivuje ON/OFF
   END_IF;
   xL^.vaz        := 0;
   xL^.fvz        := 0;
   CASE xU^.o[xU^.n].fn OF
      59:   _Nh_Web_CMD_Screen(obj := 1);                      // zoznam FAV
      41:   _Nh_Web_CMD_Screen(obj := 2);                      // sivy FAV = vazby
     198:   _Nh_Web_CMD_Screen(obj := 3);                      // Quick menu = vazby FAV
     199:   _Nh_Web_CMD_Screen(obj := 4);                      // DASH = vazby FAV
      16:   _Nh_Web_CMD_Screen(obj := 5);                      // ROMS

//            xF^.cf.c       := 1;
//            xF^.dev.n[1]   := 1;

      20:   _Nh_Web_CMD_Screen(obj := 6);                      // ZONES
     10:    _Nh_Web_CMD_Screen(obj := 7);                      // setup menu             sivy CATS
     27:    _Nh_Web_CMD_Screen(obj := 8);                      // sivy ACT
     29:    _Nh_Web_CMD_Screen(obj := 9);                      // sivy ACN
    196:    _Nh_Web_CMD_Screen(obj :=20);                      // sivy BLK
    295:    _Nh_Web_CMD_Screen(obj :=21);                      // sivy TIM
    235:    _Nh_Web_CMD_Screen(obj :=56);                      // sivy MSG

//    297:    _Nh_Web_CMD_Screen(obj :=22);                      // sivy SMW

(*
    196:    _Nh_Web_CMD_CmdScreen(obj :=15);                      // sivy BLK
    295:    _Nh_Web_CMD_CmdScreen(obj :=16);                      // sivy TIM
    297:    _Nh_Web_CMD_CmdScreen(obj :=17);                      // sivy SMW
*)
   END_CASE;
END_FUNCTION

{ $ END_IF }

//    VYKONANIE AKCIE PODLA CMD VACSINOU PREPNUTIE DO INEJ OBRAZOVKY/BROWSU

{ $ IFDEF __NH_WEB }

FUNCTION _Nh_Web_CMD    : BOOL
   VAR_IN_OUT

//      m           :  NH_M;

   END_VAR
   VAR_TEMP
      ok          : BOOL;
      yz          : SINT;
   END_VAR
   _Nh_Web_CMD   := true;
   IF xA^.tch.cmd < 255 THEN
      cmd        := 0;
      delay      := 0;
      _NhxLvl();
   END_IF;

   CASE xA^.tch.cmd OF
      0: ;

     99: // pridat specialne novu vetu v browse
            yIO := xF^.cf;
            WHILE true DO
               x := _NhFindDel(wh := 0, cx := 35, new := true);
               y := _NhFindDel(wh := 2, cx := 2,  new := true);
               IF aCfg[xF^.cf.c].par > 0 THEN
                  z := _NhFindDel(wh := 1, cx := aCfg[xF^.cf.c].par,  new := true);
               ELSE
                  z := 1;
               END_IF;
               IF x > 0 AND y > 0 AND z > 0 THEN
                  _NhxDev(c := 35, n := x, x:=18);  xDev^.ok.ok := true;
                  _NhxVaz(cv :=  2, nd := y);  xVaz^.ok.ok := true;
                  xVaz^.in.c := 35;
                  xVaz^.in.n := x;
                  xVaz^.ou   := yIO;
                  IF aCfg[xF^.cf.c].par > 0 THEN
                     _NhxPar(cp := aCfg[xF^.cf.c].par, np := z ,x:=246);  xPar^.ok.ok := true;
                     xVaz^.ou.p := z;
                  END_IF;
                  EXIT;
               ELSE
                  _Nh_Go_DbxToMem(ram := true, dbx := false );          // v 1.iteracii sa neuklada do dbx, lebo este sa budu zapisovat data
               END_IF;
            END_WHILE;
            xM^.wht        := 30;                                    // nova veta ma byt na konci browsu

    100: // prebieha editovanie nazvu  alebo pridavanie vety (editacia)

            IF xM^.new = -1   THEN                                      // CANCEL
               xM^.Naz     := xL^.Naz;                                  // do editacneho pola preberie aktualny nazov
               xM^.wht     := -1;                                       // len prekreslenie, nie nove data
            ELSIF xM^.naz <> xL^.naz AND xM^.new = 1 THEN               // uspesna modifikacia
               xL^.naz := xM^.naz;
               xM^.edt := false;
               IF xL^.obj = 2 THEN                                      // browser FAV, zmenit nazov user-fav v FAV-LIST
                  _NhFavNaz(sav := true);
               ELSE
                  _NhxCfg(c := xF^.cf.c, n := xF^.cf.n, x:=26);              // xDev,xCfg,xPar pre aktualny riadok
                  xDev^.cf.Name  := xL^.naz;
               END_IF;
               xM^.wht     := 25;

            ELSIF xM^.naz <> '' AND xM^.new = 2 THEN                       // pridanie zaznamu
                  yLVL           := xL^;
                  xM^.wht        := 30;                                    // nova veta ma byt na konci browsu
                  xU^.o[8].fn    := 49;                                    // ak by bo filter na ON, zrusi sa
                  IF xF^.cf.c = 2 THEN                                     // v niektorej kategorii sa pridava
                     CASE xF^.cf.n OF                                      // kat:2/n=5(kurenie/chladenie)
                        5 :   yIO.c :=  6;                                 // KOMFORT = pridanie regulatora
                        4 :   yIO.c := 47;                                 // VETRANIE = pridanie regulatora
                     END_CASE;
                  ELSIF xL^.obj = 5 THEN                                   // nova miestnost
                     yIO.c :=  1;
                  ELSIF xL^.obj = 47 THEN                                   // nova SVA do DALI
                     yIO.c :=  11;
                  ELSIF xL^.obj = 32 THEN                                  // nova akcia od alarmu
                     yIO.c 	:= 48;
							yCfg.rec := xF^.cf.n;											// zapamata sa cislo zony (yCfg sa vyuziva len v _Nh_INI)
                  ELSE
                     CASE xF^.cf.c OF                                      // z browsu vazieb sa pridava SCN
                         1:   yIO.c := 4;
                       ELSE   yIO.c := xF^.cf.c;
                     END_CASE;
                  END_IF;
                  yIO.n   := 0;                                            // sem pride cislo vety DEV
                  yIO.p   := 0;                                            // sem pride cislo pripadnej vety PAR
                  FOR yz := 1 TO 2 DO                                      // ak sa v 1 iteracii nenajde DEL-veta, pripadne DEL-parameter, v 2.iteracii prida nove DEL-vety, ktore sa uz najdu
                     ok3 := false;
                     IF aCfg[yIO.c].par > 0 THEN
//                       ok3   :=  aPar[ aCfg[yIO.c].par ].grp = false;      //
                         ok3   :=  true;      //9.5.23 - nove SCN s parametrom gr nopridavalo do SCN
                     END_IF;
                     IF ok3  THEN                                          // pridava sa aj parameter, nie je skupinovy
                        IF yIO.p = 0 THEN                                  // ochrana, ak by bola 2.iteracia a v prvej by sa veta nasla, uz mame je cislo
                           yIO.p := _NhFindDel(wh := 1, cx := aCfg[yIO.c].par, new := true);    // hlada sa DEL parameter, ak sa najde oznaci sa
                       END_IF;

                     END_IF;
                     IF yIO.n = 0 THEN                                     // ochrana, ak by bola 2.iteracia a v prvej by sa veta nasla, uz mame je cislo
                        yIO.n := _NhFindDel(wh := 0, cx := yIO.c, new := true);
                     END_IF;
                     IF yIO.n > 0 AND (yIO.p > 0 OR ok3 = false) THEN
                        ok3   := true;
                        CASE yIO.c OF                                   // podla hlavicky sa zisi co sa pridava
                           1 :   // ROM
                                 xRom           := xDel;
                                 xRom^.cf.rom   := 1;		//INT_TO_USINT(yIO.n);
                                 xRom^.cf.idx   := yIO.n;
                                 xRom^.cf.typ   := 1;                      // default je vnutorna zona
                                 xRom^.cf.Name  := xM^.naz;
                                 xRom^.cf.ID    := INT_TO_STRINGF(yIO.n,'%03d');
											// prida poi
											_Nh_POI_INI_NEW(cf:=yIO.c, nd1:=yIO.n, nd2:=yIO.n);

                           3 :   // zona
                                 xZon           := xDel;
                                 xZon^.cf.idx   := yIO.n;
                                 xZon^.cf.typ   := 3;                      // vnutorna zona
                                 xZon^.cf.Name  := xM^.naz;
											xZon^.cf.Rom   := _NhDefHom;  				// zona ma cislo svojho domceka

                           4 :   // SCN vseobecna, aj s ROM
                                 xScn 				:= xDel;
                                 xScn^.cf.idx   := yIO.n;
                                 xScn^.cf.Name  := xM^.naz;
                                 xScn^.cf.par   := yIO.p;                  // zona ma aj parameter
											IF xF^.cf.c = 2 THEN
												 xScn^.cf.rom   := MAX(1,_NhDefRom);
											ELSE
												xScn^.cf.rom   := xF^.rom;
											END_IF;
(*
											IF xF^.rom = 0 THEN
	                                 xScn^.cf.rom   := MAX(1,_NhDefRom);
											ELSe
	                                 xScn^.cf.rom   := MAX(1,xF^.rom);
   										END_IF;
*)
                           5 :   // ACT vseobecna, vzdy setup ROM
                                 xAct := xDel;
                                 xAct^.cf.idx   := yIO.n;
                                 xAct^.cf.Name  := xM^.naz;
											xAct^.cf.rom   := MAX(1,_NhDefHom);
//                                 xAct^.cf.rom   := INT_TO_USINT( MAX(1,MIN(xF^.cf.n,aCfg[3].rec)));

                           6 :   // HEAT
                                 xHet           := xDel;
                                 xHet^.cf.idx   := yIO.n;
                                 xHet^.cf.Name  := xM^.naz;
                                 xHet^.cf.rom   := MAX(1,_NhDefRom);
                                 xHet^.cf.par   := yIO.p;
                                 xHet^.cf.cat   := INT_TO_USINT(xF^.cf.n);
											xHet^.cf.typ 	:= 0;
											// prida poi
											_Nh_POI_INI_NEW(cf:=yIO.c, nd1:=yIO.n, nd2:=yIO.n);
(*
                                 IF xHet^.cf.cat   = 4 THEN                      // vetranie
                                    xHet^.cf.typ := 1;                           // regulator vetrania
                                 ELSE
                                    xHet^.cf.typ := 0;
                                 END_IF;
*)

                          11 :   // sva
                                 xDev2 := xDel;
                                 xDev2^.cf.idx   := yIO.n;
                                 xDev2^.cf.Name  := xM^.naz;
                                 xDev2^.cf.rom   := xF^.rom;
                                 xDev2^.cf.par   := yIO.p;

                          20 :   // zoznam FAV,DSH,QUICK
                                 xFav           := xDel;
                                 xFav^.cf.idx   := yIO.n;
                                 xFav^.cf.Name  := xM^.naz;
                                 xFav^.cx.c     := xA^.usr;
                                 xFav^.cx.n     := yIO.n;
                                 xUsr^.cx.fav   := xFav^.cx;
                                 xA^.fav        := xFav^.cx;

(*
                          35 :   // BLK vseobecna, vzdy bez ROM
                                 xBlk 				:= xDel;
                                 xBlk^.cf.idx   := yIO.n;
                                 xBlk^.cf.Name  := xM^.naz;
                                 xBlk^.cf.rom   := MAX(1,_NhDefRom);
*)

                          47 :   // HEV	- vetranie
                                 xHet           := xDel;
                                 xHet^.cf.idx   := yIO.n;
                                 xHet^.cf.Name  := xM^.naz;
                                 xHet^.cf.rom   := MAX(1,_NhDefRom);
                                 xHet^.cf.par   := yIO.p;
                                 xHet^.cf.cat   := INT_TO_USINT(xF^.cf.n);
											xHet^.cf.typ 	:= 1;
											// prida poi
											_Nh_POI_INI_NEW(cf:=yIO.c, nd1:=yIO.n, nd2:=yIO.n);

                          48 :   // ACT vseobecna, vzdy setup ROM
                                 xAla := xDel;
                                 xAla^.cf.idx   := yIO.n;
                                 xAla^.cf.Name  := xM^.naz;
//                                 xAct^.cf.rom   := INT_TO_USINT( LIMIT(xF^.cf.n,1,aCfg[3].rec) );
//											xAct^.cf.typ 	:= INT_TO_SINT(aCfg[48].rec);
                                 xAla^.cf.rom   := INT_TO_USINT( xF^.cf.n );

                          50 :   // TIM vseobecna, vzdy setup ROM
                                 xTim := xDel;
                                 xTim^.cf.idx   := yIO.n;
                                 xTim^.cf.Name  := xM^.naz;
                                 xTim^.cf.rom   := MAX(1,_NhDefRom);
                                 xTim^.cf.typ   := 1;
											ok3 				:= false;											// nema parameter
                        ELSE
                        	xDev2 				:= xDel;
                         	xDev2^.cf.idx   	:= yIO.n;
                          	xDev2^.cf.Name  	:= xM^.naz;
									ok3 				:= false;											// nema parameter
                        END_CASE;
                       	xDev2 				:= xDel;
								IF xDev2^.cf.rom > 0 THEN												// ak sa nepriradila rom
									;
								ELSIF  aCfg[yIO.c].RomIsZone THEN
									xDev2^.cf.rom   := MAX(1,_NhDefHom);							// default Room
								ELSE
									xDev2^.cf.rom   := MAX(1,_NhDefRom);							// default hlavna zona / domcek
								END_IF;

                        xL^.rw1.c  := yIO.c;                                  		// pre spravny refresh
                        xL^.rw1.n  := yIO.n;;

								xDev2 := xDel;
                        _NhxUsr(u := xA^.usr );                                  	// pri vstupe do session namapuje usra, potom uz v programe nikdy
                        EXIT;
                     ELSE
                        _Nh_Go_DbxToMem(ram := true, dbx := false );          			// v 1.iteracii sa neuklada do dbx, lebo este sa budu zapisovat data
                     END_IF;
                  END_FOR;
            ELSE
               RETURN;
            END_IF;
            xM^.edt     := false;
            xU^.o[1] := xM^.mno[1];
            xU^.o[2] := xM^.mno[2];
            xM^.wht        := 30;                                    // nova veta ma byt na konci browsu

    101: // vstup do modifikacie nazvu alebo pridanie novej vety cez nazov

            xM^.new := 1;                                         // znak pridavania vety
            IF xF^.rom > 0 THEN
               _NhxRom(nr := xF^.rom,x:=-5);
            END_IF;
            IF xM^.edt = false THEN                                  // pridanie
               IF xL^.obj = 47 THEN                                  // pridanie SVA
                  xM^.naz := xL^.Naz;
               ELSE
                  xM^.naz := '';
               END_IF;
               xM^.edt := true;
               xM^.new := 2;                                         // znak pridavania vety
            ELSE

               xM^.naz := xL^.naz;
            END_IF;

            yTx1 := xM^.naz;
            REPLACE_CHAR(c1:=16#01,c2:=16#00,input:=yTx1);           // vyhodenie znaku SOH {Start Of Header}
            xM^.naz :=yTx1;

            xM^.mno[1]  := xU^.o[1];                                 // zalohovanie m1
            xM^.mno[2]  := xU^.o[2];
            xU^.o[1].fn := 46;                                    // CANCEL vlavo hore
            xU^.o[1].cm := 100;                                   // CANCEL vlavo hore
            xU^.o[2].fn := 0;
            cmd         := 100;
            xM^.wht     := -1;                                     // len prekreslenie, nie nove data

     102: // VYMAZAT ZAZNAM
            _NhxDev(c := xR^.h.cf.c, n:= xR^.h.cf.n, x:=19);                                   // namapuje vetu aby sme odcitali cf,nd
            yVaz.in  := xR^.h.cf;
            yVaz.ou  := xR^.h.cf;                                                               // pre SCN/FAV-list
				If xA^.usr = 1 THEN
            	vi      	:= xR^.h.cf.c;
	            rmp      := 1;
   	         xM^.wht  := 0;
      		ELSE
					vi  			:= 255;
					rmp			:= 255;
   	         xM^.wht  	:= 10;
				END_IF;
            CASE vi OF
              1 : // ROM
						_Nh_POI_INI_NEW(cf:=xR^.h.cf.c, nd1:=xR^.h.cf.n, nd2:=xR^.h.cf.n, del:=true);

              3 : // ZON
                  xZon     := xDev;
						ii			:=	INT_TO_USINT(xR^.h.cf.n);
	               FOR nd := 1 TO aCfg[1].rec DO
							//PRERADIT rom do DEFAULT domceka
							IF _NhxPt(c:=1, n := nd,x:=-123) THEN
			               IF xPt^.cf.rom = ii THEN
									xPt^.cf.rom := MAX(1,_NhDefHom);
								END_IF;
							END_IF;
            	   END_FOR;

              4: 	// DEL SCN
						;
//  _NhfVaz(vaz := 3, row := false, whf := 3, del := true, all := true);           // aVaz[2] - SCN list  in+ou , kde je ACT
              5: // DEL ACT
						;
//                  _NhfVaz(vaz := 4, row := false, whf := 3, del := true, all := true);          // IO : in+ou , kde je ACT

//             35 : // DEL BLK
//                  _NhfVaz(vaz := 1, row := false, whf := 2, del := true, all := true);          // zoznam FAV, k SCN, sCN je v ou
//                  _NhfVaz(vaz := 2, row := false, whf := 3, del := true, all := true);          // IO : in+ou , kde je ACT

              6: // HET
						_Nh_POI_INI_NEW(cf:=xR^.h.cf.c, nd1:=xR^.h.cf.n, nd2:=xR^.h.cf.n, del:=true);

//                  _NhfVaz(vaz := 1, row := false, whf := 2, del := true, all := true);          // zoznam FAV, k HET ou
//                  _NhfVaz(vaz := 2, row := false, whf := 3, del := true, all := true);          // IO : in+ou , kde je ACT

             20: // hlavicka FAV + obsah
                  xFav           := xDev;
                  yVaz.in        := xFav^.cx;
                  xUsr^.cx.fav   := xFav^.cx;
                  _NhfVaz(vaz := 1, row := false, whf := 1, del := true, all := true);          // zoznam FAV, k hlavicke, hlavicka je v in
                  // usrovi nastavi FAV-ALL
                  _NhxDev(c := 20, n:= 4, x:=19);                                              // oblubene vsetkych
                  xFav           := xDev;
                  xA^.fav        := xFav^.cx;
                  xUsr^.cx.fav   := xFav^.cx;

           	  40:	// TGL
						;
              46 : // MSG  - zmazat aj vaz[] = zoznam usrov, ktori dostanu SMS
                  xM^.wht  := 0;
                  rmp  		:= 0;

              47 : // HEV
						_Nh_POI_INI_NEW(cf:=xR^.h.cf.c, nd1:=xR^.h.cf.n, nd2:=xR^.h.cf.n, del:=true);
(*

             39 : // RFID card
                  _NhfVaz(pg := 133,  wh := 2, all := true);                   // vymaze vsetky vazby tohto oblubeneho ()
                  _NhDelRec(cf := xR^.h.cf.c, nd := xR^.h.cf.n);                  // vymaze zaznam
*)
//            ELSE
//                  xM^.wht  := 10;                                                                // nic sa nevymazalo, refresh dat od 1.riadku
//                  rmp      := 1;

             255 : // not acces right
		   			;
				END_CASE;
				IF rmp = 1 THEN
               _NhfVaz(vaz := 1, row := false, whf := 2, del := true, all := true);          // zoznam FAV, k HET ou
               _NhfVaz(vaz := 2, row := false, whf := 3, del := true, all := true);          // IO : in+ou WSB,TLA..PIR
               _NhfVaz(vaz := 3, row := false, whf := 3, del := true, all := true);          // IO : in+ou, vazby sCN
               _NhfVaz(vaz := 4, row := false, whf := 3, del := true, all := true);          // IO : in+ou, vazby ACT
            END_IF;
            IF xM^.wht = 0 THEN
               _NhxCfg(c := xR^.h.cf.c, n:= xR^.h.cf.n, x:=57);                                      // koli parametru
               IF xDev^.cf.par > 0 THEN
                  _NhFindDel(wh := 1, cx := aCfg[xR^.h.cf.c].par, nx := xDev^.cf.par, ok := false ); // vymazat parameter
               END_IF;
               _NhFindDel(wh := 0, cx := xR^.h.cf.c, nx := xR^.h.cf.n, ok := false );           // vymazat samotnu vetu aj jej pripadne parametre
               xM^.wht := 15;                                                                   // refresh pre vymazanu vetu
            END_IF;
            xM^.new     := 0;
            xA^.tch.cpy := 0;
            xA^.tch.del := 0;

     103: // kopirovat VETU VAZBY a ZOSORTOVAT
            xM^.wht := 10;
            IF _NhfVaz(vaz := 2, whf := 10) THEN                                             // najde vetu vaz, ktora odpoveda riadku. AJ S PARAMTRAMI
               nd    := nDel+1;                                                              // nova veta by mala byt fyzicky za kopirovanou vetou
               yVaz  := xVaz^;                                                               // data kopirovanej vety
               yIO   := yVaz.ou;                                                             // zapamatanie zdroja DEV najma parametra
               nDel  := _NhFindDel(wh := 2, cx := 2, new := false, ok := false);             // skusi najst DEL-vetu vazby
               nDel  := _NhNewVaz(ok := nDel > 0, par := true, vaz := 2, nv := nDel);
               IF yIO.p > 0 AND yVaz.ou.p > 0  THEN
                  rb := _NhCpyRec(wh := 1,cf := aCfg[yIO.c].par ,ns := yIO.p, nd :=yVaz.ou.p);  // prekopiruje parameter
               END_IF;
               IF nDel > 0 THEN
                  _NhSrtVaz(vaz := 2, poz := nd, new := nDel);
//                  _NhSrtVaz(poz := nd, new := nDel);
                  xM^.wht  := 25;
               END_IF;
	            xM^.new     := 0;
   	         xA^.tch.cpy := 0;
      	      xA^.tch.del := 0;
            END_IF;

      1: // potiahnutie dolu
            xM^.wht        := 1;
            cmd := 0;         ///***
//            xA^.tch.cm     := 1;

      2: // potiahnutie hore
            xM^.wht        := 2;
            cmd := 0;         ///***
//            xA^.tch.cm     := 2;

      3: // POTIAHNUTIE DOLAVA = DELETE/COPY
            xM^.wht := 0;
            IF xL^.dsh <> 1                  THEN                 // del iba dsh = 1
               ;
            ELSIF xA^.tch.row = 0               THEN
               ;
            ELSIF xR^.h.cf.c = 0                THEN
               ;
            ELSIF xL^.obj = 50 AND xR^.h.chk    THEN                 // kopirovanie vazby
               // obmedzit !! co sa da kopirovat
                xM^.new     := SINT_TO_INT(xA^.tch.row);
                xA^.tch.cpy := true;
                xM^.wht     := 10;                                    // prekreslenie dat bez vytvorenia indexu

            ELSIF aCfg[xR^.h.cf.c].del THEN
               xM^.wht     := 10;                                    // prekreslenie dat bez vytvorenia indexu
               _NhxDev(c := xR^.h.cf.c, n := xR^.h.cf.n, x:=20);
               IF xR^.h.cf.c = 20 THEN                    					// zoznam skupin FAV
                  IF xR^.h.cf.n  > 4 THEN                               // prve 4 sa nezmazavaju
                     xFav := xDev;
                     IF xM^.set = false THEN
                        xM^.wht := 0;
                     ELSIF xFav^.cx.c <> xA^.usr THEN
                        xM^.wht := 0;
                     END_IF;
                  ELSE
                     xM^.wht     := 0;                                    // prekreslenie dat bez vytvorenia indexu
                  END_IF;
               ELSIF xR^.h.cf.c = 4 OR xR^.h.cf.c = 5 THEN                // SCN, ACT
                  If xA^.usr = 1 OR xUsr^.cx.ZonList[ xDev^.cf.rom ] THEN
                     ;
                  ELSE
                     xM^.wht := 0;
                  END_IF;
               ELSIF xA^.usr <> 1                  THEN
                  xM^.wht     := 0;
               ELSIF xR^.h.cf.c = 3 AND xR^.h.cf.n < 4 THEN                // zony
                  xM^.wht := 0;
               END_IF;
               IF xM^.wht = 10 THEN
                  xM^.new     := SINT_TO_INT(xA^.tch.row);					// toto rozhoduje
                  xA^.tch.del := true;
               END_IF;
            END_IF;

      4: // potiahnutie doprava
            xM^.wht     := -1;
      5: // neznamy prikaz - sposoboval rozhodenie obrazovky, posun o lvl dopredu a xL^.obj := 0
            xM^.wht     := -1;
      6: // press bez CMD
            xM^.wht     := -1;
     20:    _Nh_Web_CMD_Action(mnu := 0);                                              // HOME screen
     21:    _Nh_Web_CMD_Action(mnu := 4);                                              // FAV
     22:    _Nh_Web_CMD_Action(mnu := 5);                                              // ROOMS
     23:    _Nh_Web_CMD_Action(mnu := 6);                                              // CATS
     24:    _Nh_Web_CMD_Action(mnu := 7);                                              // ACT/SCN/TIM/BLK/SMW

     25: // SETUP MENU (z ikony NachHouse)
            _Nh_Web_CMD_Action(mnu := 1);

     26: // filter ON/OFF
            IF xF^.cf.c = 1 THEN
               CASE xU^.o[8].fn OF
                  49 : xU^.o[8].fn := 51;              // OFF (52)--> ON
                  51 : xU^.o[8].fn := 57;              // Pohyb
                 ELSE  xU^.o[8].fn := 49;              // off
               END_CASE;
            ELSE
               CASE xU^.o[8].fn OF
                  49 : xU^.o[8].fn := 51;              // OFF (52)--> ON
                    ELSE  xU^.o[8].fn := 49;              // off
               END_CASE;
            END_IF;
            xM^.wht  := 20;                        // nove data

     27: // ZMENA OBLUBENEHO
            _NhxDev2(c := xR^.h.cf.c, n := xR^.h.cf.n, x:=21);  // NAMAPUJE riadok
            xFav     := xDev2;
            xA^.fav  := xFav^.cx;
(*
            _NhxUsr(u := xA^.usr);
            CASE xA^.fav.n OF
              -1: xA^.fav.c := _Nh_U12(xUsr^.cx.OwnDsh,xA^.usr,1);
                  xUsr^.cx.dsh := xA^.fav;
              -2: xA^.fav.c := _Nh_U12(xUsr^.cx.OwnQck,xA^.usr,1);
                  xUsr^.cx.qck := xA^.fav;
            ELSE  xUsr^.cx.fav := xA^.fav;
            END_CASE;
*)
            xUsr^.cx.fav := xA^.fav;
            xU^.n   := 4;                                            // podhodi, ze bolo predtym stlacene menu FAV
            _Nh_Web_CMD_Action(mnu := 4);                                     // este raz stlaci menu FAV aby sa preplo na nieco ine

     28: // PREPNI STAV ON/OFF na DEV
            IF xL^.obj = 0 THEN                                      // HOME QUICK
               _NhxCfg(c := xO^.cf.c, n := xO^.cf.n, x:=62);                 // xDev,xCfg,xPar
            ELSE
               _NhxCfg(c := xR^.h.cf.c, n := xR^.h.cf.n, par := true, p := xR^.h.cf.p, x:=29);  // xDev,xCfg,xPar
            END_IF;
            IF xL^.psn THEN														// len u ZON/ROM
					xDev^.al.in.cmd := 55;
//					xRom	:= xDev;

(*
					IF xO^.cf.c = 3 THEN												// zona zamyka svoje miestnosti
						xRom^.al.in.cmd := 55; 							         // LOCK/UNLOCK
					ELSIF xRom^.cx.lck.stat > 0 THEN
						xRom^.cx.lck.stat 	:= 0;
						xRom^.cx.lck.et   	:= 0;
					ELSE
						xRom^.cx.lck.stat 	:= 1;
						xRom^.cx.lck.et   	:= MAX(xRom^.cx.lck.tdOu,1);
					END_IF;
*)
(*
					IF xRom^.cx.lck.stat > 0 THEN
						xRom^.cx.lck.what := 2;												// odomkni
					ELSE
						xRom^.cx.lck.what := 1;		                           	// zamkni
					END_IF;

							IF xRom^.cx.lck.stat < 6 THEN
								xRom^.cx.lck.stat := xRom^.cx.lck.stat + 1;
							ELSE
								xRom^.cx.lck.stat := 0;
							END_IF;
                     xRom^.cx.lck.et := 13;
*)

            ELSIF xR^.h.cf.c = 15 THEN                                        // PIR - vysle testovaci signal
               IF xM^.set THEN
                  xDev^.al.in.cmd   := 21;                                 // z webu vysle testovaci signal
                  xDev^.al.in.par   := xR^.h.cf.p;
               END_IF;

            ELSIF xR^.h.cf.c = 35 THEN                                     // BLK
               xDev^.al.in.cmd   := 1;                                     // prepni

//            ELSIF xR^.h.cf.c = 44 THEN                                     // DLg
//               xDev^.al.in.cmd   := 1;                                     // prepni

            ELSIF xR^.h.cf.c = 22 THEN                                     // Prepnut usra

//               aWeb.A[1].usr :=  SINT_TO_USINT(xA^.tch.row);
//               _NhxUsr(u := xA^.usr );                                  // pri vstupe do session namapuje usra, potom uz v programe nikdy
//               aWeb.A[1].fav  := xUsr^.cx.fav;

            ELSIF xR^.h.chk THEN                                           // ovplyvnuje len parmeter vazby - pri vybratej vazbe sa zmeni LVL v parametri
              	IF xPar^.all.lvl > 0 THEN
                 xPar^.all.lvl   := 0;
               ELSIF xDev^.al.ou.Val > 0.0 THEN
                  xPar^.all.lvl   := REAL_TO_USINT(xDev^.al.ou.Val);
//		         ELSIF aCfg[xR^.h.cf.c].lvl254 THEN
//                  xPar^.all.lvl   := 254;
               ELSE
                  xPar^.all.lvl   := 100;
               END_IF;
               IF xL^.vis  THEN                                            // ak je vis zapne/vypne sa ale neulozi sa do default parametra z webu
                  xDev^.al.in.cmd 	:= 14;
                  xDev^.al.in.par   := xR^.h.cf.p;
               END_IF;
            ELSE
               xDev^.al.in.cmd   := 1;                                     // prepni bez oneskorenia
               xDev^.al.in.par   := 0;                                     // pri takomto zadani sa zoberie default parameter
            END_IF;
            xA^.tch.End       := true;                                     //ukoncenie vyhodnocovanie pres
            xM^.wht           := 0;                                        // v tomto cykle sa nepokracuje do browsu, lebo sa nastavuje DEV , az v druhom cykle
            cmd               := 251;                                      // aby sa vratilo do browsu po nastaveni

     29: // ZAPNI (AKCIU)
            _NhxCfg(c := xR^.h.cf.c, n := xR^.h.cf.n, x:=30);  // xDev,xCfg,xPar
            xDev^.al.in.cmd := 11;
            xDev^.al.in.par := 0;                                        // pri takomto zadani sa zoberie default parameter
            xM^.wht         := -1;                                       // len prekreslenie riadkov, nie nove data

     30: // >>  O UROVEN DOPREDU Z RIADKA
         CASE xR^.h.cf.c OF
           0 : ;	// _NheLvl( lvl := 0 );
         ELSE
         	IF _NheLvl( lvl := 1 ) = false THEN                            // o LVL dopredu
          		xA^.tch.cmd := 0;
           		RETURN;
          	END_IF;
         END_CASE;
			IF xF^.cf.c <> 2 THEN
	         _NhxDev(c := xF^.cf.c ,n := xF^.cf.n, x:=631);
			END_IF;
         CASE xF^.cf.c OF
            1:
					IF xM^.lvd[xM^.lvl-1].obj = 14 THEN                      // ide sa do 1.ROM z browsu zon SEC
                  _Nh_Web_CMD_Screen(obj := 15);                                    // >> 1 ROM/SEC
               ELSE
                  _Nh_Web_CMD_Screen(obj := 10);                                    // >> 1 ROM
               END_IF;
            2: CASE xF^.cf.n OF                                         // hlbsie do podkategorii
//                 6 : _Nh_Web_CMD_Screen(obj := 13);                                 // >> 1 CAT = SEC
                41 : _Nh_Web_CMD_Screen(obj := 49);                                 // >> zoznam DALI master
               ELSE  _Nh_Web_CMD_Screen(obj := 12);                                 // >> 1 CAT (ostatne)
               END_CASE;
            3:
               _Nh_Web_CMD_Screen(obj := 11);                                 // >> 1 ZONE
         ELSE
            xM^.lvl     := xM^.lvl-1;
            xA^.tch.cmd := 0;
            RETURN;
         END_CASE;

     31: // <  O UROVEN SPAT
         _NheLvl(lvl:=-1);                                              // o LVL dopredu
         xM^.htt :=  '';

     32: // SETUP O UROVEN DOPREDU Z RIADKA
         IF _NheLvl(lvl:=1) THEN                      // o LVL dopredu bez prebratia menu
            _Nh_Web_CMD_Screen(obj := 50,obr:=xR^.o.ob[1].fn, eMnu:=1 );                        // VAZBY,LIST....
         END_IF;

     33: // CHECK SPODNE MENU VAZIEB ON/OFF  - vo vazbach
            _Nh_Vaz_CHK(chg:=true );
            xM^.wht := 20;
     34 :   // zmena kategorie
            xM^.wht := 20;
            _Nh_Vaz_CAT(chg:=true);
     35: // ROM: ALL / 1.rom
            xM^.wht := 20;
            _Nh_Vaz_ROM(chg:=true);

     36: // VISIBLE  - vo vazbach
            xU^.o[6].fn :=  _Nh_O12(xU^.o[6].fn = 112,113,112);
            xL^.vis := xU^.o[6].fn = 113;                                     // vsetko prestavovanie prenasat do HW ()
            xM^.wht := 25;                                                     // refresh od 1.riadka s novymi datatmi do riadkov

     37: // prepnut na SCN,ACT-LIST
            _Nh_Web_CMD_Screen(obj := 51);                        // LIST....
            xM^.wht := 20;

     38: // prepnut na PLAY (IO) v SCN/ACT
            _Nh_Web_CMD_Screen(obj := 50);                        // VAZBY,LIST....
            xM^.wht := 20;

     39: // prepnut filter ROM v browse 1.ZONE
         xL^.fvz := NOT xL^.fvz;                               // pri clicku zmeni
         IF xL^.fvz THEN
            xF^.rom := INT_TO_USINT(xF^.cf.n);
            xU^.o[1].fn := 38;
         ELSE
            xF^.rom := 0;
            xU^.o[1].fn := 36;
         END_IF;
         xM^.wht := 20;

     40: // priradit FAV z riadku
            _NhfVaz(vaz := 1, new := xR^.o.ob[3].fn <> 43, del := xR^.o.ob[3].fn = 43, par := false);
            xM^.wht := 25;

     41: // CHECK z riadku - priradit/vymazat vazby aVaz[2]

				aSys.RefCycNew		:=	1;												// zabezpeci vymazanie OWN a aktualizaciu vstupoc
             xM^.wht     	:= 25;

            IF xR^.h.cf.c > 0 THEN                                                           // ochrana pre Err
               _NhxPt(c := xF^.cf.c, n := xF^.cf.n,x:=55);
               xDev2       := xPt;
               _NhxPt(c := xR^.h.cf.c, n := xR^.h.cf.n,x:=48);
               xDev        := xPt;
               yIdxR.dev   := xR^.h.cf;                           // potrebne pre _NhChkRoM
            END_IF;

            IF xR^.h.cf.c = 0 OR xR^.h.cf.c > _Nh_CFG THEN                                                           // ochrana pre Err
               yTx2     := CONCAT('ERR!-01 VAZ _NhBrwMenu 41:CHECK z riadku. xR^.h.cf.c/n/p: ',
                                    USINT_TO_STRING(xR^.h.cf.c),'/',INT_TO_STRING(xR^.h.cf.n),'/',INT_TO_STRING(xR^.h.cf.p));
               _Nh1RowTxt(logRst := 1, adTime := 3);
            ELSIF _Nh_Chk_IODev(set := true) THEN             // vo vazbe je ROM ... kde sa inak priradzuje ako pri VAZ
//				ELSIF _Nh_Chk_SCN(set := true) THEN	;
                           ;
//				{$IFDEF __NH_DALI}
         	   ELSIF _Nh_Chk_DALI(set := true) THEN ;           // vazbe DLg -> DLs  ... kde sa inak priradzuje ako pri VAZ
//			   {$END_IF}

            ELSIF xL^.vaz  = 3 THEN
               IF xR^.h.chk THEN
                  _NhfVaz(del := true, vaz := xL^.vaz, whf := 10);               // vymaze sa veta  hladana aj s parametrami
               ELSE
                  xR^.h.in := false;
                  _NhfVaz(new := true, vaz := xL^.vaz);
               END_IF;

            ELSIF xL^.vaz  = 4 THEN
               IF xR^.h.chk THEN
                  _NhfVaz(del := true, vaz := xL^.vaz);               // vymaze sa veta  hladana aj s parametrami
               ELSE
                  xR^.h.in := false;
                  _NhfVaz(new := true, vaz := xL^.vaz);
               END_IF;

            ELSIF xR^.h.chk = false  THEN
               xR^.h.in := _NhFilDev(wht:=5, row:=xR^.h.cf.c, n:=xF^.cf.c);
               _NhfVaz(new := true, vaz := xL^.vaz);
               ok := true;
               _NhxCfg (c := xVaz^.in.c, n := xVaz^.in.n, par := true, p := xVaz^.in.p, x:=61 );         // namapuje In s parametrom
               _NhxCfg2(c := xVaz^.ou.c, n := xVaz^.ou.n, par := true, p := xVaz^.ou.p, x:=67 );         // namapuje Ou s parametrom
//               IF xVaz^.in.c = 13 OR xVaz^.in.c = 14 OR xVaz^.in.c = 40 THEN                                // prednastavi CMD do clickov vo WSB
               IF aCfg[xVaz^.in.c].tgrp = 13 THEN                                // prednastavi CMD do clickov vo WSB
                  ok    := false;
                  cmd   := 0;
                  pWsb := xPar;
                  xWsb := xDev;
						_Nh_Get_Frm260(cmd := true, cf := xVaz^.ou.c, nd := xVaz^.ou.n, grp := aCfg[ xVaz^.ou.c ].mWsb );
               ELSIF xVaz^.in.c = 15 THEN                                              // PIR

//                  xPar2^.out.Delay := 30;

               ELSIF xF^.cf.c = 6 THEN                                               // KURENIE

//                  xDev2^.cf.typ  := USINT_TO_SINT(xVaz^.in.c);
//                  IF _Nh_ADD_FIL_BRW(cf := xF^.cf.c, typ := xDev2^.cf.typ ) THEN
//                    xDev2^.cf.rom  := xDev^.cf.rom ;
//                    xF^.rom        := xDev2^.cf.rom;
//                    xU^.o[5].fn    := 18;                                             // filter miestnosti na 1.rom
//                  END_IF;

               END_IF;
               IF ok AND xVaz^.ou.p > 0 AND aCfg[xVaz^.ou.c].ou  THEN                  // ak nebolo WSB a len pre vystupne DEV
                  yIO    := xVaz^.ou;
                  _NhxCfg (c := yIO.c, n := yIO.n, x:=35);                                  // este raz Dev, bez parametra
                  _NhxPar(cp := aCfg[yIO.c].par, np := xDev^.cf.par,x:=-1014);                 // zisti default paramter, kde je aktualny stav
                  _NhxCfg2(c := yIO.c, n := yIO.n, par := true, p := yIO.p, x:=36 );       // namapuje novy parameter
                  IF xDev^.al.ou.val > 0.0   THEN                                      // dev aktualne ON
                     i  := 0;
                     CASE yIO.c OF
                       0 : ;
                       4 : yIO.c := 0;																	// SCN
                      10 : i := 1;                                             			// SVD
                      11 : i := 2;                                                     // SVA
                      12 : i := 3;																		// RGB
							 		xPar2^ := xPar^;                                            // do parametra vlozi aktualny stav pre RGB moze cely par
                      21 : i := 1;                                                     // ZAS
                     END_CASE;
                     CASE i OF                                                         // skupinove vlastnosti
                       1 : //SVD,SVA,ZAS
                           xPar2^.all := xPar^.all;                                    // defult casy
                       2 : //SVD,SVA,ZAS
                           xPar2^.all := xPar^.all;                                    // defult casy
                           xPar2^.sva := xPar^.sva;                                    // defult casy
                     END_CASE;
	                  xPar2^.all.lvl  	:= REAL_TO_USINT(xDev^.al.ou.val);
//						ELSIF acfg[yIO.c].Lvl254 THEN
//	                  xPar2^.all.lvl  	:= 254;
 						ELSE
       					xPar2^.all.lvl  	:= 100;
            		END_IF;
//                  IF xVaz^.in.c = 15 AND i > 0 THEN                                 	// PIR oproti OUT, ktore ma PAR
                  IF xVaz^.in.c = 15 THEN                                 					// PIR oproti OUT, ktore ma PAR
                     xPar2^.all.tOff 		:= 450;                                      // default cas 45s
                     xPar2^.all.BlPirOff 	:= 0;														// sam pir sa neblokuje
                     xPar2^.all.BlPirOn  	:= 0;
                  END_IF;
               END_IF;
               xL^.rw1 := xR^.h.cf;
            ELSE
(*
               _Nh_Chk_RoW(chk:=false,vaz:=true);
               IF xF^.cf.c = 6 THEN                                               // KURENIE
                  _NhxDev2(c := xF^.cf.c, n := xF^.cf.n, x:=59 );         // namapuje Ou s parametrom
                  IF _Nh_ADD_FIL_BRW(cf := xF^.cf.c, typ := xDev2^.cf.typ, set:=false ) THEN
                     xDev2^.cf.typ := 0;
                     xDev2^.cf.rom  := 0 ;
                     IF xF^.rom = 0 THEN
                        xU^.o[5].fn    := 17;                                             // filter miestnosti na 1.rom
                     END_IF;
                  END_IF;
               END_IF;

*)

               _Nh_Chk_RoW(chk:=false,vaz:=true);
               _NhfVaz(del := true, vaz := xL^.vaz, whf := 10);               // vymaze sa veta  hladana aj s parametrami
            END_IF;

     42: // LED na WSB ON/OFF
            _NhxDev(c := xR^.h.cf.c, n := xR^.h.cf.n, x:=21);                      // pre zistenie xCfg toho co je v hlacivke (DEV alebo SCN), ACT sem vobec nepride
            xDev^.al.in.cmd   := 17;                                          // prepni LED
            xDev^.al.in.par   := SINT_TO_INT(xA^.tch.obj-5);                  // 1.led je v objekte 5
            cmd      := 252;
            xM^.wht  := -1;
//            xA^.tch.cmd       := 252;                                         // ked sa vrati, len prekresli browser
//            RETURN;

     43: // zmena zobrazenia riadok - dash
//            rb := _NhBrwDsh(chg := true, mnu := SINT_TO_USINT(xA^.tch.obj));

            rb       := _Nh_Brw_Dsh_Chg(chg := true, mnu := xL^.obd);
            xM^.wht  := 20;                                                      // prekreslenie browsu + nove data

     44: // zrusenie beziaceho OFF-casu nad DEV/PIR
				IF _NhxDev2(c := xR^.h.cf.c, n := xR^.h.cf.n, x:=23 ) THEN
					IF xR^.h.cf.c = 15 THEN														// PIR
		            IF _NhxRom(nr := xDev2^.cf.rom, x:=23 )THEN                 // rom, kde je PIR
		               xRom^.me.BlPirOff 	:= 0;
				      END_IF;
					ELSE
            		xDev2^.al.et   := 0;                                        // po case vypnut
//  		          xDev2^.al.ex   := 0;                                       // celkovy cas zapnutia
					END_IF;
					_NhDevRef(xR  := xDev2);
				END_IF;
            xM^.wht        := -1;                                             // len prekreslenie, nie nove data

     45: // zrusenie blokovania PIR v miestnosti

            _NhxDev2(c := xR^.h.cf.c, n := xR^.h.cf.n, x:=23 );                    // xDev,xCfg,xPar pre aktualny riadok
            IF _NhxRom(nr:=xDev2^.cf.rom, x:=-12) THEN
               xRom^.me.BlPirOn 		:= 0;
               xRom^.me.BlPirOff 	:= 0;
					_NhDevRef(xR  := xDev2);
            END_IF;
            xM^.wht        := -1;                                             // len prekreslenie, nie nove data

     46: // CHECK z riadku - priradit ROM
            xM^.wht := 10;
            _NhxDev(c := xF^.cf.c, n := xF^.cf.n, x:=327);
            IF xR^.h.chk = false THEN
               IF xDev^.cf.rom > 0 THEN
                  _NhxDev2(c := 1, n := xR^.h.cf.n, x:=427);
                  yTx2  := CONCAT(xDev2^.cf.ID,' ',xDev2^.cf.Name);
                  yTx2  := LEFT(yTx2,20);
               END_IF;
               ok             := xDev^.cf.rom <> INT_TO_USINT(xR^.h.cf.n);
               xDev^.cf.rom   := INT_TO_USINT(xR^.h.cf.n);                  // priradi novy ROM
               CASE xF^.cf.c OF
                 13 : xDev^.al.rmp := 1;                                   // vypne stlacenie
                 14 : xDev^.al.rmp := 1;
                 43 : // DLs
                     // pri zmene uklada
//                     yTx3 := CONCAT(_Nh_ADR_ROT,'/CFG/_',USINT_TO_STRINGF(43,'%03d'),'.DEV');
//                     _NhVarSdc(src := PTR_TO_UDINT(xDev), siz := UINT_TO_UDINT(aCfg[43].Siz) * 128   );
               END_CASE;
               rb             := _NhSysUpd();
            END_IF;

     47:    _Nh_Web_CMD_Action(mnu := 5);                                              // ROOMS

     48:   // ROL - prepni slider ROL/LAM

         _NhxDev(c := xR^.h.cf.c, n := xR^.h.cf.n, x:=66 );
         xRol              := xDev;
         xRol^.cx.SetLam   := NOT xRol^.cx.SetLam;                            // robi sa to inak v procedure, ale ked nasleduje wht=25, tak tu
         xR^.o.ob[6].BgC   := _Nh_U12(xRol^.cx.SetLam,2,3);
         xM^.wht 				:= 25;

     49:   // BRA - zafixovat zatvorene
         _NhxDev(c := xR^.h.cf.c, n := xR^.h.cf.n, x:=29 );
         xGat := xDev;
         IF xGat^.cx.btn THEN 								//
            xGat^.al.in.CMD := 50;                       // potvrdit otvorene
			ELSE
            xGat^.al.in.CMD := 51;                     	// potvrdit zatvorene
         END_IF;
         xM^.wht           := -1;

     50: // odskok z Home screen DEV/CAT/ROM

         yIO  := xB^.r[ xA^.tch.row ].o.ob[xA^.tch.obj].cf;
         _NheBrw(wht := 6);
	   	xU^.o[3]    := eMnH.o[3];                                     // aktivuje HOME
		   xU^.o[8]    := eMnH.o[8];                                     // aktivuje ON/OFF
			xF^.cf 		:= yIO;
         CASE xF^.cf.n OF                                         // hlbsie do podkategorii
//           6 :	_Nh_Web_CMD_Screen(obj := 13);                                 // >> 1 CAT = SEC
           6 :	xL^.psn  := true;
			  		_Nh_Web_CMD_Screen(obj :=  6);                                 // >> 1 CAT = SEC
          41 : _Nh_Web_CMD_Screen(obj := 49);                                 // >> zoznam DALI master
         ELSE  _Nh_Web_CMD_Screen(obj := 12);                                 // >> 1 CAT (ostatne)
         END_CASE;

     51: // >>  do podkategorie
    		IF _NheLvl(lvl:=1) = false THEN                            // o LVL dopredu
    			xA^.tch.cmd := 0;
     			RETURN;
       	END_IF;
         CASE xF^.cf.n OF
           41:  _Nh_Web_CMD_Screen(obj := 49);                                 // >> zoznam DALI master
           ELSE  _Nh_Web_CMD_Screen(obj := 12);                                 // >> 1 CAT (ostatne)
         END_CASE;

     52:   // ROL - zafixovat zatvorene
         _NhxDev(c := xF^.cf.c, n := xF^.cf.n, x:=63 );
         xDev^.al.in.cmd    := 52;
         xM^.wht           := -1;

     53:   // ROL - zafixovat otvorene
         _NhxDev(c := xF^.cf.c, n := xF^.cf.n, x:=33 );
         xDev^.al.in.cmd := 53;
         xM^.wht           := -1;

     60:    // HOME - objekty
            CASE   xB^.r[xA^.tch.row].o.ob[xA^.tch.obj].fn OF
             87 : // pir
                  xU^.o[8].fn := 57;
                  _Nh_Web_CMD_Action(mnu := 5);
            ELSE
            ;
            END_CASE;
            xM^.wht           := 25;

     63: // spodne menu xU[3] CHECK - CH2 zapnut=vypnut iba priradene : DLg
         xM^.wht := 20;                                                    // nove data
         IF xF^.cf.c = 43 THEN                                             // hed:DLS -> DLg:row
            xL^.fvz := NOT xL^.fvz;
            IF xL^.fvz THEN
               xF^.rom := 0;
            END_IF;
			ELSE
            xL^.fvz := NOT xL^.fvz;
         END_IF;
         xU^.o[3].fn    := _Nh_O12(xL^.fvz,38,35);

     64: // spodne menu xU[4] vacsinou CAT
         xM^.wht := -1;                                                    // nove data

     65: // spodne menu xU[5] MIESTNOSTI
     66: // spodne menu xU[6] visible
     67: // spodne menu xU[8] List DEV
     68: // spodne menu xU[9] PLAY/ ON*OFF...

(*
     54: // aktivovat/deaktivovat blikac/opozdovac pre DEV  (pridat/odobrat vetu v acfg[36])

            xPar^.out.Bl1 := NOT xPar^.out.Bl1;
            IF xPar^.out.Bl1 THEN                                // treba najst vetu
               xPar^.out.BlX := _NhFindDel(wh:=0, cx:=36, new:=true, nOk :=true);
               IF xPar^.out.BlX = 0 THEN
                  xPar^.out.BlX := aCfg[36].rec + 1;
                  _NhDbxRam(ram := true, dbx := false );          // v 1.iteracii sa neuklada do dbx, lebo este sa budu zapisovat data
               END_IF;
            ELSIF xPar^.out.BlX > 0 THEN                         // vymazat
               _NhFindDel(cx:=36, nx :=xPar^.out.BlX, ok:=0,new:=0);
               xPar^.out.BlX := 0;
            END_IF;
            xM^.wht := 30;                                       // v tomto cykle sa nepokracuje do browsu, lebo sa nastavuje DEV , az v druhom cykle
*)
(*

     59: // akcie menu - filtre pre priradenie miestnosti
          xM^.wht := -1;
         IF xF^.cf.c = 43 THEN                                          // hlavicke je DLS, riadky DLg
            CASE xA^.tch.obj OF
//              2 : xL^.dsh := _Nh_U12(xL^.dsh = 3,1,3);                  // DSH
              3 : xU^.o[3].fn := _Nh_O12(xU^.o[3].fn = 35,38,35);       // len s priradenym DEV
                  xM^.wht := 20;
//              4 : // cat
              8 : xU^.o[8].fn := _Nh_O12(xU^.o[8].fn = 49,51,49);       // ON/OFF
            ELSE
               xM^.wht := 25;
            END_CASE;
         END_IF;
*)

     69: // zmena modu nastavit pridanie RFID karty / hladanie
            _NhxDev(c := 38, n := 1, x:=34 );                                   // nastavit sa na RFID snimac vratnicovy
            IF xU^.o[2].fn = 32 THEN
               xU^.o[2].fn       := 47;                                    // obrazok + na zelenom = pridanie karty
               xDev^.al.in.cmd   := 102;
            ELSE
               xU^.o[2].fn       := 32;                                    // hladanie karty
               xDev^.al.in.cmd   := 101;
            END_IF;
            xM^.wht := -1;                                     // len prekreslenie, nie nove data

     74: // prepnut v spodnom menu na RBBWA
         IF _NheLvl(lvl:=1) THEN
            _Nh_Web_CMD_Screen(obj := 56,obr:=xR^.o.ob[1].fn,eMnu:=1);
         END_IF;
     75: // prepnut v spodnom menu na RGBWA
     		_Nh_Web_CMD_Screen(obj := 56, n := SINT_TO_USINT(xA^.tch.obj));
